(* IEC 61131-3 sources: Automated-Water-Pump/build, 2 files *)

(* ---- plc.st ---- *)
TYPE
  LOGLEVEL : (CRITICAL, WARNING, INFO, DEBUG) := INFO;
END_TYPE

FUNCTION_BLOCK LOGGER
  VAR_INPUT
    TRIG : BOOL;
    MSG : STRING;
    LEVEL : LOGLEVEL := INFO;
  END_VAR
  VAR
    TRIG0 : BOOL;
  END_VAR

  IF TRIG AND NOT TRIG0 THEN
  {{
   LogMessage(GetFbVar(LEVEL),(char*)GetFbVar(MSG, .body),GetFbVar(MSG, .len));
  }}
  END_IF;
  TRIG0:=TRIG;
END_FUNCTION_BLOCK

FUNCTION_BLOCK python_eval
  VAR_INPUT
    TRIG : BOOL;
    CODE : STRING;
  END_VAR
  VAR_OUTPUT
    ACK : BOOL;
    RESULT : STRING;
  END_VAR
  VAR
    STATE : DWORD;
    BUFFER : STRING;
    PREBUFFER : STRING;
    TRIGM1 : BOOL;
    TRIGGED : BOOL;
  END_VAR

  {extern void __PythonEvalFB(int, PYTHON_EVAL*);__PythonEvalFB(0, data__);}
END_FUNCTION_BLOCK

FUNCTION_BLOCK python_poll
  VAR_INPUT
    TRIG : BOOL;
    CODE : STRING;
  END_VAR
  VAR_OUTPUT
    ACK : BOOL;
    RESULT : STRING;
  END_VAR
  VAR
    STATE : DWORD;
    BUFFER : STRING;
    PREBUFFER : STRING;
    TRIGM1 : BOOL;
    TRIGGED : BOOL;
  END_VAR

  {extern void __PythonEvalFB(int, PYTHON_EVAL*);__PythonEvalFB(1,(PYTHON_EVAL*)(void*)data__);}
END_FUNCTION_BLOCK

FUNCTION_BLOCK python_gear
  VAR_INPUT
    N : UINT;
    TRIG : BOOL;
    CODE : STRING;
  END_VAR
  VAR_OUTPUT
    ACK : BOOL;
    RESULT : STRING;
  END_VAR
  VAR
    py_eval : python_eval;
    COUNTER : UINT;
    _TMP_ADD10_OUT : UINT;
    _TMP_EQ13_OUT : BOOL;
    _TMP_SEL15_OUT : UINT;
    _TMP_AND7_OUT : BOOL;
  END_VAR

  _TMP_ADD10_OUT := ADD(COUNTER, 1);
  _TMP_EQ13_OUT := EQ(N, _TMP_ADD10_OUT);
  _TMP_SEL15_OUT := SEL(_TMP_EQ13_OUT, _TMP_ADD10_OUT, 0);
  COUNTER := _TMP_SEL15_OUT;
  _TMP_AND7_OUT := AND(_TMP_EQ13_OUT, TRIG);
  py_eval(TRIG := _TMP_AND7_OUT, CODE := CODE);
  ACK := py_eval.ACK;
  RESULT := py_eval.RESULT;
END_FUNCTION_BLOCK

PROGRAM program0
  VAR
    EmStop : BOOL;
    E1 : BOOL;
    E2 : BOOL;
    P1 : BOOL;
    P2 : BOOL;
  END_VAR
  VAR
    _TMP_AND50_OUT : BOOL;
    _TMP_NOT44_OUT : BOOL;
    _TMP_OR46_OUT : BOOL;
    _TMP_AND51_OUT : BOOL;
  END_VAR

  _TMP_AND50_OUT := AND(NOT(E2) AND NOT(E1), NOT(EmStop));
  P2 := _TMP_AND50_OUT;
  _TMP_NOT44_OUT := NOT(NOT(E1));
  _TMP_OR46_OUT := OR(NOT(E2) AND NOT(E1), NOT(E2) AND _TMP_NOT44_OUT);
  _TMP_AND51_OUT := AND(NOT(EmStop), _TMP_OR46_OUT);
  P1 := _TMP_AND51_OUT;
END_PROGRAM

CONFIGURATION Config0

  RESOURCE Res0 ON PLC
    TASK task0(INTERVAL := T#20ms,PRIORITY := 0);
    PROGRAM instance0 WITH task0 : program0;
  END_RESOURCE
END_CONFIGURATION

(* ---- generated_plc.st ---- *)
PROGRAM program0
  VAR
    EmStop AT %IX0.1 : BOOL;
    E1 AT %IX0.2 : BOOL;
    E2 AT %IX0.3 : BOOL;
    P1 AT %QX0.0 : BOOL;
    P2 AT %QX0.1 : BOOL;
  END_VAR
  VAR
    _TMP_AND50_OUT : BOOL;
    _TMP_NOT44_OUT : BOOL;
    _TMP_OR46_OUT : BOOL;
    _TMP_AND51_OUT : BOOL;
  END_VAR

  _TMP_AND50_OUT := AND(NOT(E2) AND NOT(E1), NOT(EmStop));
  P2 := _TMP_AND50_OUT;
  _TMP_NOT44_OUT := NOT(NOT(E1));
  _TMP_OR46_OUT := OR(NOT(E2) AND NOT(E1), NOT(E2) AND _TMP_NOT44_OUT);
  _TMP_AND51_OUT := AND(NOT(EmStop), _TMP_OR46_OUT);
  P1 := _TMP_AND51_OUT;
END_PROGRAM

CONFIGURATION Config0

  RESOURCE Res0 ON PLC
    TASK task0(INTERVAL := T#20ms,PRIORITY := 0);
    PROGRAM instance0 WITH task0 : program0;
  END_RESOURCE
END_CONFIGURATION
